# EPICS autosave request: dxp/branches/R3-0-branch/dxpApp/Db/xMAP_settings.req
$(P)CollectMode
$(P)PixelAdvanceMode
$(P)PixelsPerRun
$(P)PixelsPerBuffer
$(P)IgnoreGate
$(P)SyncCount
$(P)InputLogicPolarity
